(* IEC 61131-3 sources: repolevel_ST_code_completion/ground_truth/repoeval_PID_controller/readful_result, 2 files *)

(* ---- Tank.st ---- *)
It seems like you have provided multiple fragments of the same code from the `Tank.st` file located in the `PID_controller-Models` directory. The code appears to define a `FUNCTION_BLOCK` called `Tank`, which simulates the behavior of a tank that fills and empties based on input and output flow rates (`Process_In` and `Process_Out`). The tank's level is updated periodically based on the `SampleTime` input, and the level is constrained between `Lower_limit` and `Upper_limit`.

Here is a consolidated version of the provided code:

```st
// A.J. Jaworowski 2015-02-20
// Simulering av en tank med RedBull
FUNCTION_BLOCK Tank
VAR_INPUT
	Process_In: REAL;  // Flöde in per sekund, testa vad som händer on du matar in 100
					   // Därefter ska regulatorns OUT in i denna ingång.
	Process_Out: REAL; // Flöde ut per sekund, typ 90
					   // Effekten blir att tanken fylls med 10 per sekund
					   // Full efter ca 1 minut - testa
	SampleTime: TIME;  // Uppdateringstid, typ 100ms
	Lower_limit: REAL; // Tankens lägsta nivå, typ 0
	Upper_limit: REAL; // Tankens max nivå, kanske 500
END_VAR
VAR_OUTPUT
	Level: REAL; // Nivån i tanken
END_VAR
VAR
	now: TIME;
	lastTime: TIME;
	proc_sum_in: REAL := 0;
	proc_sum_out: REAL := 0;
	temp: REAL;
	millis: UINT := 1000;
	proc_out: REAL;
END_VAR

// Logic to update the tank level
now := TIME();
IF ((now - lastTime) > SampleTime) THEN
	Level := Level + TIME_TO_REAL(SampleTime) / millis * (Process_In - Process_Out);
	IF Level < Lower_limit THEN
		Level := Lower_limit;
	END_IF;
	IF Level > Upper_limit THEN
		Level := Upper_limit;
	END_IF;
	lastTime := now;
END_IF;
```

### Explanation of the Code:
1. **Inputs (`VAR_INPUT`)**:
   - `Process_In`: The inflow rate of the tank (e.g., liters per second).
   - `Process_Out`: The outflow rate of the tank.
   - `SampleTime`: The time interval for updating the tank level.
   - `Lower_limit`: The minimum level of the tank.
   - `Upper_limit`: The maximum level of the tank.

2. **Outputs (`VAR_OUTPUT`)**:
   - `Level`: The current level of the tank.

3. **Internal Variables (`VAR`)**:
   - `now`: The current time.
   - `lastTime`: The last time the tank level was updated.
   - `proc_sum_in` and `proc_sum_out`: Variables to track cumulative inflow and outflow (not fully implemented in the provided code).
   - `temp`: A temporary variable (not used in the provided code).
   - `millis`: A constant representing the number of milliseconds in a second (1000).
   - `proc_out`: Another temporary variable (not used in the provided code).

4. **Logic**:
   - The tank level is updated periodically based on the `SampleTime` interval.
   - The new level is calculated using the formula:
     ```
     Level := Level + (SampleTime in seconds) * (Process_In - Process_Out)
     ```
   - The level is then constrained between `Lower_limit` and `Upper_limit`.
   - The `lastTime` variable is updated to the current time after each update.

### Notes:
- The code appears to be written in Structured Text (ST), a programming language used in industrial automation and control systems.
- The comments in the code are in Swedish, and they provide additional context for the variables and logic.
- Some variables (`proc_sum_in`, `proc_sum_out`, `temp`, `proc_out`) are declared but not used in the provided code. If they are not used elsewhere in the file, they can be removed to clean up the code.
- The `TIME_TO_REAL` function is used to convert the `SampleTime` from a `TIME` data type to a `REAL` (floating-point) value for calculations.

Let me know if you need further clarification or assistance!

(* ---- Tank_1.st ---- *)
It seems like you have provided multiple fragments of the same code from the `Tank.st` file located in the `PID_controller-Models` directory. The code appears to define a `FUNCTION_BLOCK` called `Tank`, which simulates the behavior of a tank that fills and empties based on input and output flow rates (`Process_In` and `Process_Out`). The tank's level is updated periodically based on the `SampleTime` input, and the level is constrained between `Lower_limit` and `Upper_limit`.

Here is a consolidated version of the provided code:

```st
// A.J. Jaworowski 2015-02-20
// Simulering av en tank med RedBull
FUNCTION_BLOCK Tank
VAR_INPUT
	Process_In: REAL;  // Flöde in per sekund, testa vad som händer on du matar in 100
					   // Därefter ska regulatorns OUT in i denna ingång.
	Process_Out: REAL; // Flöde ut per sekund, typ 90
					   // Effekten blir att tanken fylls med 10 per sekund
					   // Full efter ca 1 minut - testa
	SampleTime: TIME;  // Uppdateringstid, typ 100ms
	Lower_limit: REAL; // Tankens lägsta nivå, typ 0
	Upper_limit: REAL; // Tankens max nivå, kanske 500
END_VAR
VAR_OUTPUT
	Level: REAL; // Nivån i tanken
END_VAR
VAR
	now: TIME;
	lastTime: TIME;
	proc_sum_in: REAL := 0;
	proc_sum_out: REAL := 0;
	temp: REAL;
	millis: UINT := 1000;
	proc_out: REAL;
END_VAR

// Logic to update the tank level
now := TIME();
IF ((now - lastTime) > SampleTime) THEN
	Level := Level + TIME_TO_REAL(SampleTime) / millis * (Process_In - Process_Out);
	IF Level < Lower_limit THEN
		Level := Lower_limit;
	END_IF;
	IF Level > Upper_limit THEN
		Level := Upper_limit;
	END_IF;
	lastTime := now;
END_IF;
```

### Explanation of the Code:
1. **Inputs (`VAR_INPUT`)**:
   - `Process_In`: The inflow rate of the tank (e.g., liters per second).
   - `Process_Out`: The outflow rate of the tank.
   - `SampleTime`: The time interval for updating the tank level.
   - `Lower_limit`: The minimum level of the tank.
   - `Upper_limit`: The maximum level of the tank.

2. **Outputs (`VAR_OUTPUT`)**:
   - `Level`: The current level of the tank.

3. **Internal Variables (`VAR`)**:
   - `now`: The current time.
   - `lastTime`: The last time the tank level was updated.
   - `proc_sum_in` and `proc_sum_out`: Variables to track cumulative inflow and outflow (not fully implemented in the provided code).
   - `temp`: A temporary variable (not used in the provided code).
   - `millis`: A constant representing the number of milliseconds in a second (1000).
   - `proc_out`: Another temporary variable (not used in the provided code).

4. **Logic**:
   - The tank level is updated periodically based on the `SampleTime` interval.
   - The new level is calculated using the formula:
     ```
     Level := Level + (SampleTime in seconds) * (Process_In - Process_Out)
     ```
   - The level is then constrained between `Lower_limit` and `Upper_limit`.
   - The `lastTime` variable is updated to the current time after each update.

### Notes:
- The code appears to be written in Structured Text (ST), a programming language used in industrial automation and control systems.
- The comments in the code are in Swedish, and they provide additional context for the variables and logic.
- Some variables (`proc_sum_in`, `proc_sum_out`, `temp`, `proc_out`) are declared but not used in the provided code. If they are not used elsewhere in the file, they can be removed to clean up the code.
- The `TIME_TO_REAL` function is used to convert the `SampleTime` from a `TIME` data type to a `REAL` (floating-point) value for calculations.

Let me know if you need further clarification or assistance!
